PROGRAM MAIN
VAR
END_VAR

END_PROGRAM

(* stored: Version 1.1.0.1
   POU MAIN: Id {5d58acb1-82c9-4411-9ef5-68ff26592bf1} *)
